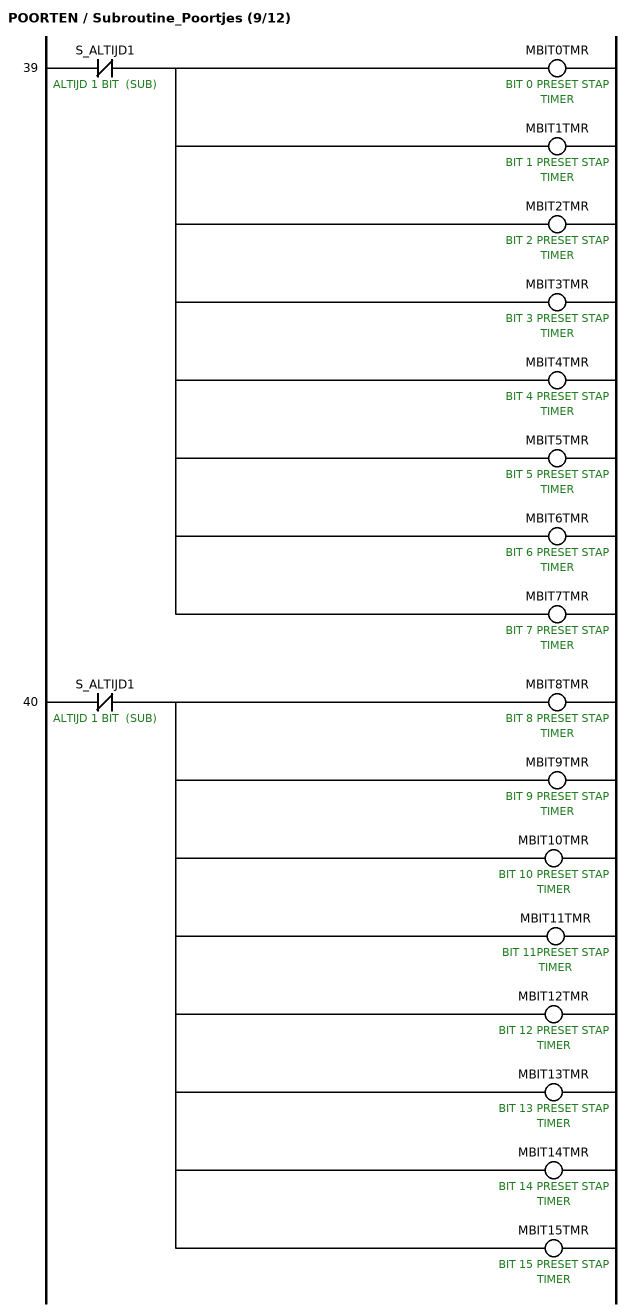
; [picture p493: POORTEN / Subroutine_Poortjes, rungs 39-40]
; rung 39
LDNOT S_ALTIJD1  ; ALTIJD 1 BIT  (SUB)
OUT MBIT0TMR  ; BIT 0 PRESET STAP TIMER
OUT MBIT1TMR  ; BIT 1 PRESET STAP TIMER
OUT MBIT2TMR  ; BIT 2 PRESET STAP TIMER
OUT MBIT3TMR  ; BIT 3 PRESET STAP TIMER
OUT MBIT4TMR  ; BIT 4 PRESET STAP TIMER
OUT MBIT5TMR  ; BIT 5 PRESET STAP TIMER
OUT MBIT6TMR  ; BIT 6 PRESET STAP TIMER
OUT MBIT7TMR  ; BIT 7 PRESET STAP TIMER
; rung 40
LDNOT S_ALTIJD1  ; ALTIJD 1 BIT  (SUB)
OUT MBIT8TMR  ; BIT 8 PRESET STAP TIMER
OUT MBIT9TMR  ; BIT 9 PRESET STAP TIMER
OUT MBIT10TMR  ; BIT 10 PRESET STAP TIMER
OUT MBIT11TMR  ; BIT 11PRESET STAP TIMER
OUT MBIT12TMR  ; BIT 12 PRESET STAP TIMER
OUT MBIT13TMR  ; BIT 13 PRESET STAP TIMER
OUT MBIT14TMR  ; BIT 14 PRESET STAP TIMER
OUT MBIT15TMR  ; BIT 15 PRESET STAP TIMER

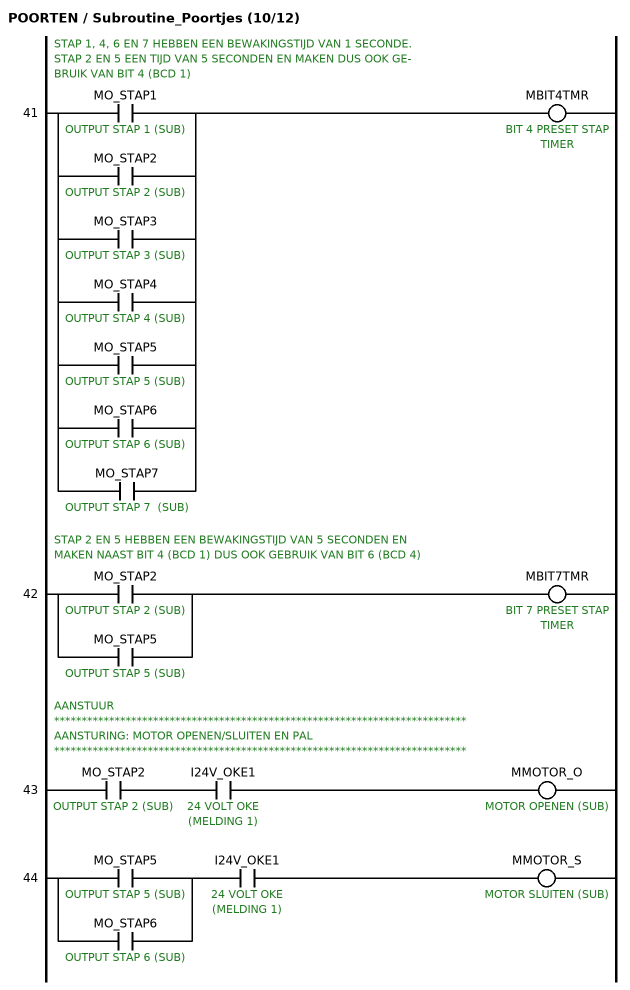
; rung 41: STAP 1, 4, 6 EN 7 HEBBEN EEN BEWAKINGSTIJD VAN 1 SECONDE. / STAP 2 EN 5 EEN TIJD VAN 5 SECONDEN EN MAKEN DUS OOK GE- / BRUIK VAN BIT 4 (BCD 1)
LD MO_STAP1  ; OUTPUT STAP 1 (SUB)
OR MO_STAP2  ; OUTPUT STAP 2 (SUB)
OR MO_STAP3  ; OUTPUT STAP 3 (SUB)
OR MO_STAP4  ; OUTPUT STAP 4 (SUB)
OR MO_STAP5  ; OUTPUT STAP 5 (SUB)
OR MO_STAP6  ; OUTPUT STAP 6 (SUB)
OR MO_STAP7  ; OUTPUT STAP 7  (SUB)
OUT MBIT4TMR  ; BIT 4 PRESET STAP TIMER
; rung 42: STAP 2 EN 5 HEBBEN EEN BEWAKINGSTIJD VAN 5 SECONDEN EN / MAKEN NAAST BIT 4 (BCD 1) DUS OOK GEBRUIK VAN BIT 6 (BCD 4)
LD MO_STAP2  ; OUTPUT STAP 2 (SUB)
OR MO_STAP5  ; OUTPUT STAP 5 (SUB)
OUT MBIT7TMR  ; BIT 7 PRESET STAP TIMER
; rung 43: AANSTUUR / *************************************************************************** / AANSTURING: MOTOR OPENEN/SLUITEN EN PAL / ***************************************************************************
LD MO_STAP2  ; OUTPUT STAP 2 (SUB)
AND I24V_OKE1  ; 24 VOLT OKE (MELDING 1)
OUT MMOTOR_O  ; MOTOR OPENEN (SUB)
; rung 44
LD MO_STAP5  ; OUTPUT STAP 5 (SUB)
OR MO_STAP6  ; OUTPUT STAP 6 (SUB)
AND I24V_OKE1  ; 24 VOLT OKE (MELDING 1)
OUT MMOTOR_S  ; MOTOR SLUITEN (SUB)

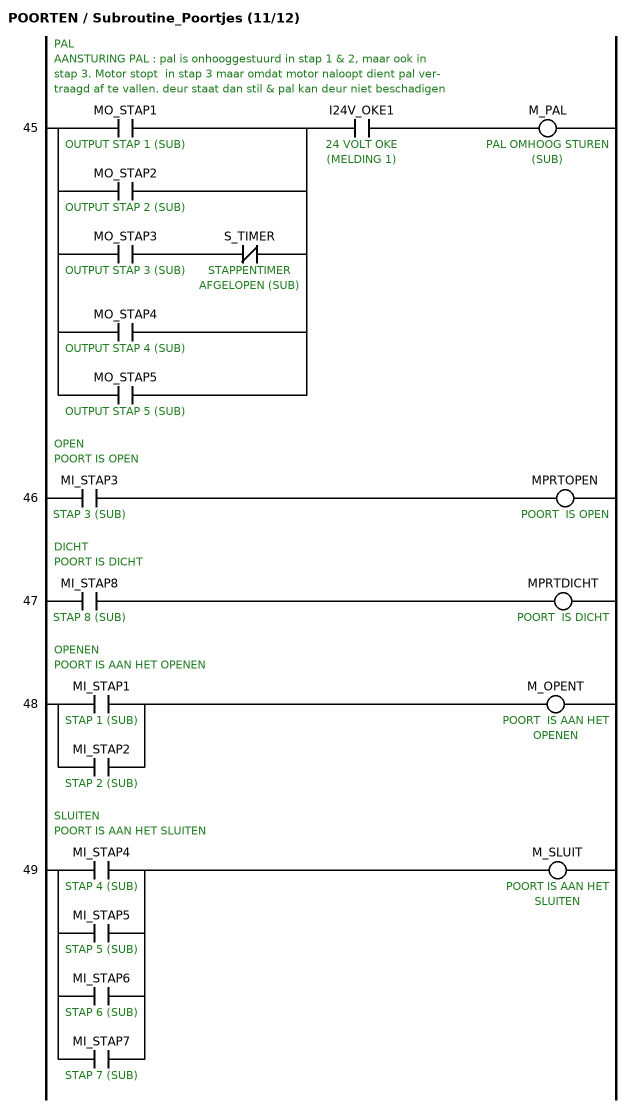
; rung 45: PAL / AANSTURING PAL : pal is onhooggestuurd in stap 1 & 2, maar ook in / stap 3. Motor stopt  in stap 3 maar omdat motor naloopt dient pal ver- / traagd af te vallen. deur staat dan stil & pal kan deur niet beschadigen
LD MO_STAP1  ; OUTPUT STAP 1 (SUB)
OR MO_STAP2  ; OUTPUT STAP 2 (SUB)
LD MO_STAP3  ; OUTPUT STAP 3 (SUB)
ANDNOT S_TIMER  ; STAPPENTIMER AFGELOPEN (SUB)
ORLD
OR MO_STAP4  ; OUTPUT STAP 4 (SUB)
OR MO_STAP5  ; OUTPUT STAP 5 (SUB)
AND I24V_OKE1  ; 24 VOLT OKE (MELDING 1)
OUT M_PAL  ; PAL OMHOOG STUREN (SUB)
; rung 46: OPEN / POORT IS OPEN
LD MI_STAP3  ; STAP 3 (SUB)
OUT MPRTOPEN  ; POORT  IS OPEN
; rung 47: DICHT / POORT IS DICHT
LD MI_STAP8  ; STAP 8 (SUB)
OUT MPRTDICHT  ; POORT  IS DICHT
; rung 48: OPENEN / POORT IS AAN HET OPENEN
LD MI_STAP1  ; STAP 1 (SUB)
OR MI_STAP2  ; STAP 2 (SUB)
OUT M_OPENT  ; POORT  IS AAN HET OPENEN
; rung 49: SLUITEN / POORT IS AAN HET SLUITEN
LD MI_STAP4  ; STAP 4 (SUB)
OR MI_STAP5  ; STAP 5 (SUB)
OR MI_STAP6  ; STAP 6 (SUB)
OR MI_STAP7  ; STAP 7 (SUB)
OUT M_SLUIT  ; POORT IS AAN HET SLUITEN

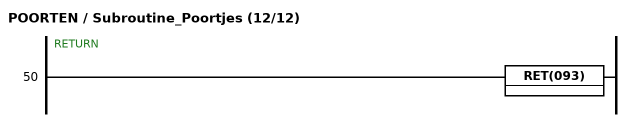
; rung 50: RETURN
RET(093)

### Section EINDE
; rung 0: PROGR_END
END(001)